TYPE FlowCalTestResult :
STRUCT
	flow : LREAL;
	weight : LREAL;
	startTime : 
END_STRUCT
END_TYPE

(* stored: Version 1.1.0.1, ProductVersion 3.1.0.36
   DUT FlowCalTestResult: Id {9c647d8e-a0cb-45bf-aff1-d518d1b8b1f0} *)
